FUNCTION SubtractionFunction : REAL
VAR_INPUT
	i_valueA : REAL;
	i_valueB : REAL;
END_VAR
VAR
END_VAR

SubtractionFunction := i_valueA - i_valueB;

END_FUNCTION

(* stored: Version 1.1.0.1, ProductVersion 3.1.4022.12
   POU SubtractionFunction: Id {3f353174-a718-498d-8032-8da49980b23c}, SpecialFunc None *)
